// TIA Portal V18 export
ORGANIZATION_BLOCK "Status Monitor"   // OB127, LAD, ProgramCycle
TITLE = Main Control block
{ S7_Optimized_Access := 'TRUE' }
AUTHOR : HenriP
VERSION : 0.1
// stored: AutoNumber true, IsIECCheckEnabled false, SetENOAutomatically false
   VAR_INPUT
      Initial_Call : Bool;   // Initial call of this OB
      Remanence : Bool;   // =True, if remanent data are available
   END_VAR
   VAR_TEMP
      ClearError : Bool;
   END_VAR
   VAR_TEMP   // added for the SCL form of the ladder/FBD networks
      _w1 : Bool;
   END_VAR
BEGIN

REGION Network 1: Monitor
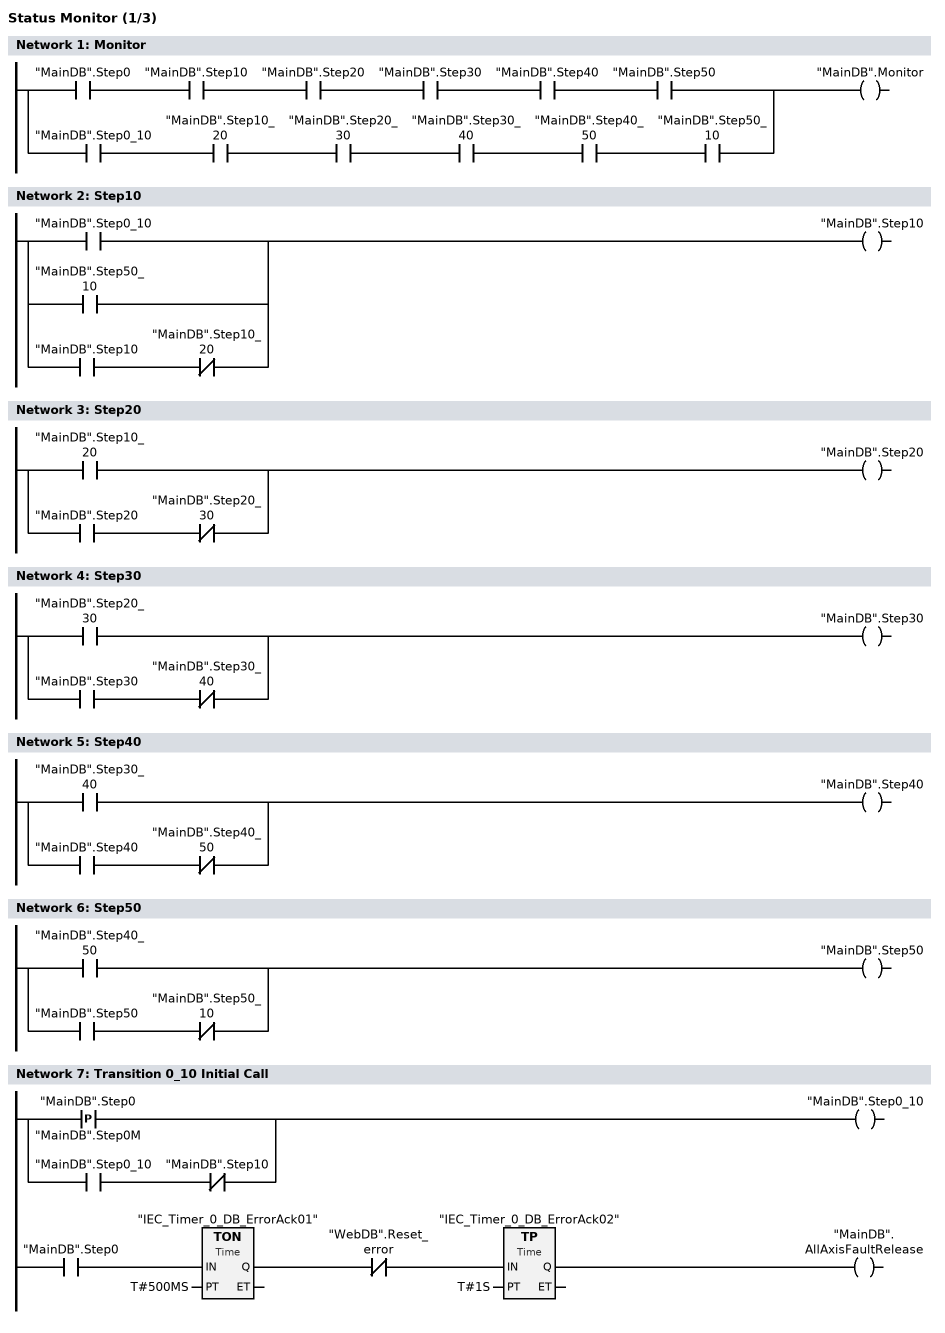
   RUNG wire#powerrail
      Contact( "MainDB".Step0 )
      Contact( "MainDB".Step10 )
      Contact( "MainDB".Step20 )
      Contact( "MainDB".Step30 )
      Contact( "MainDB".Step40 )
      Contact( "MainDB".Step50 )
      wire#w1
      Coil( "MainDB".Monitor )
   END_RUNG
   RUNG wire#powerrail
      Contact( "MainDB".Step0_10 )
      Contact( "MainDB".Step10_20 )
      Contact( "MainDB".Step20_30 )
      Contact( "MainDB".Step30_40 )
      Contact( "MainDB".Step40_50 )
      Contact( "MainDB".Step50_10 )
   END_RUNG wire#w1
   // the same network as SCL:
   "MainDB".Monitor := ("MainDB".Step0 AND "MainDB".Step10 AND "MainDB".Step20 AND "MainDB".Step30 AND "MainDB".Step40 AND "MainDB".Step50) OR ("MainDB".Step0_10 AND "MainDB".Step10_20 AND "MainDB".Step20_30 AND "MainDB".Step30_40 AND "MainDB".Step40_50 AND "MainDB".Step50_10);
END_REGION

REGION Network 2: Step10
   RUNG wire#powerrail
      Contact( "MainDB".Step0_10 )
      wire#w1
      Coil( "MainDB".Step10 )
   END_RUNG
   RUNG wire#powerrail
      Contact( "MainDB".Step50_10 )
   END_RUNG wire#w1
   RUNG wire#powerrail
      Contact( "MainDB".Step10 )
      I_Contact( "MainDB".Step10_20 )
   END_RUNG wire#w1
   // the same network as SCL:
   "MainDB".Step10 := "MainDB".Step0_10 OR "MainDB".Step50_10 OR ("MainDB".Step10 AND NOT "MainDB".Step10_20);
END_REGION

REGION Network 3: Step20
   RUNG wire#powerrail
      Contact( "MainDB".Step10_20 )
      wire#w1
      Coil( "MainDB".Step20 )
   END_RUNG
   RUNG wire#powerrail
      Contact( "MainDB".Step20 )
      I_Contact( "MainDB".Step20_30 )
   END_RUNG wire#w1
   // the same network as SCL:
   "MainDB".Step20 := "MainDB".Step10_20 OR ("MainDB".Step20 AND NOT "MainDB".Step20_30);
END_REGION

REGION Network 4: Step30
   RUNG wire#powerrail
      Contact( "MainDB".Step20_30 )
      wire#w1
      Coil( "MainDB".Step30 )
   END_RUNG
   RUNG wire#powerrail
      Contact( "MainDB".Step30 )
      I_Contact( "MainDB".Step30_40 )
   END_RUNG wire#w1
   // the same network as SCL:
   "MainDB".Step30 := "MainDB".Step20_30 OR ("MainDB".Step30 AND NOT "MainDB".Step30_40);
END_REGION

REGION Network 5: Step40
   RUNG wire#powerrail
      Contact( "MainDB".Step30_40 )
      wire#w1
      Coil( "MainDB".Step40 )
   END_RUNG
   RUNG wire#powerrail
      Contact( "MainDB".Step40 )
      I_Contact( "MainDB".Step40_50 )
   END_RUNG wire#w1
   // the same network as SCL:
   "MainDB".Step40 := "MainDB".Step30_40 OR ("MainDB".Step40 AND NOT "MainDB".Step40_50);
END_REGION

REGION Network 6: Step50
   RUNG wire#powerrail
      Contact( "MainDB".Step40_50 )
      wire#w1
      Coil( "MainDB".Step50 )
   END_RUNG
   RUNG wire#powerrail
      Contact( "MainDB".Step50 )
      I_Contact( "MainDB".Step50_10 )
   END_RUNG wire#w1
   // the same network as SCL:
   "MainDB".Step50 := "MainDB".Step40_50 OR ("MainDB".Step50 AND NOT "MainDB".Step50_10);
END_REGION

REGION Network 7: Transition 0_10 Initial Call
   RUNG wire#powerrail
      P_Contact(operand := "MainDB".Step0, bit := "MainDB".Step0M)
      wire#w1
      Coil( "MainDB".Step0_10 )
   END_RUNG
   RUNG wire#powerrail
      Contact( "MainDB".Step0_10 )
      I_Contact( "MainDB".Step10 )
   END_RUNG wire#w1
   RUNG wire#powerrail
      Contact( "MainDB".Step0 )
      { S7_Templates := "time_type := Time" } "IEC_Timer_0_DB_ErrorAck01".TON(pt := T#500MS, et =>)
      I_Contact( "WebDB".Reset_error )
      { S7_Templates := "time_type := Time" } "IEC_Timer_0_DB_ErrorAck02".TP(pt := T#1S, et =>)
      Coil( "MainDB".AllAxisFaultRelease )
   END_RUNG
   // the same network as SCL:
   #_w1 := "MainDB".Step0 AND NOT "MainDB".Step0M;   // rising edge of "MainDB".Step0
   "MainDB".Step0M := "MainDB".Step0;
   "MainDB".Step0_10 := #_w1 OR ("MainDB".Step0_10 AND NOT "MainDB".Step10);
   "IEC_Timer_0_DB_ErrorAck01".TON(IN := "MainDB".Step0, PT := T#500MS);
   "IEC_Timer_0_DB_ErrorAck02".TP(IN := "IEC_Timer_0_DB_ErrorAck01".Q AND NOT "WebDB".Reset_error, PT := T#1S);
   "MainDB".AllAxisFaultRelease := "IEC_Timer_0_DB_ErrorAck02".Q;
END_REGION

REGION Network 8: Transition10-20 Check PLC Operating State -> Wait Ready
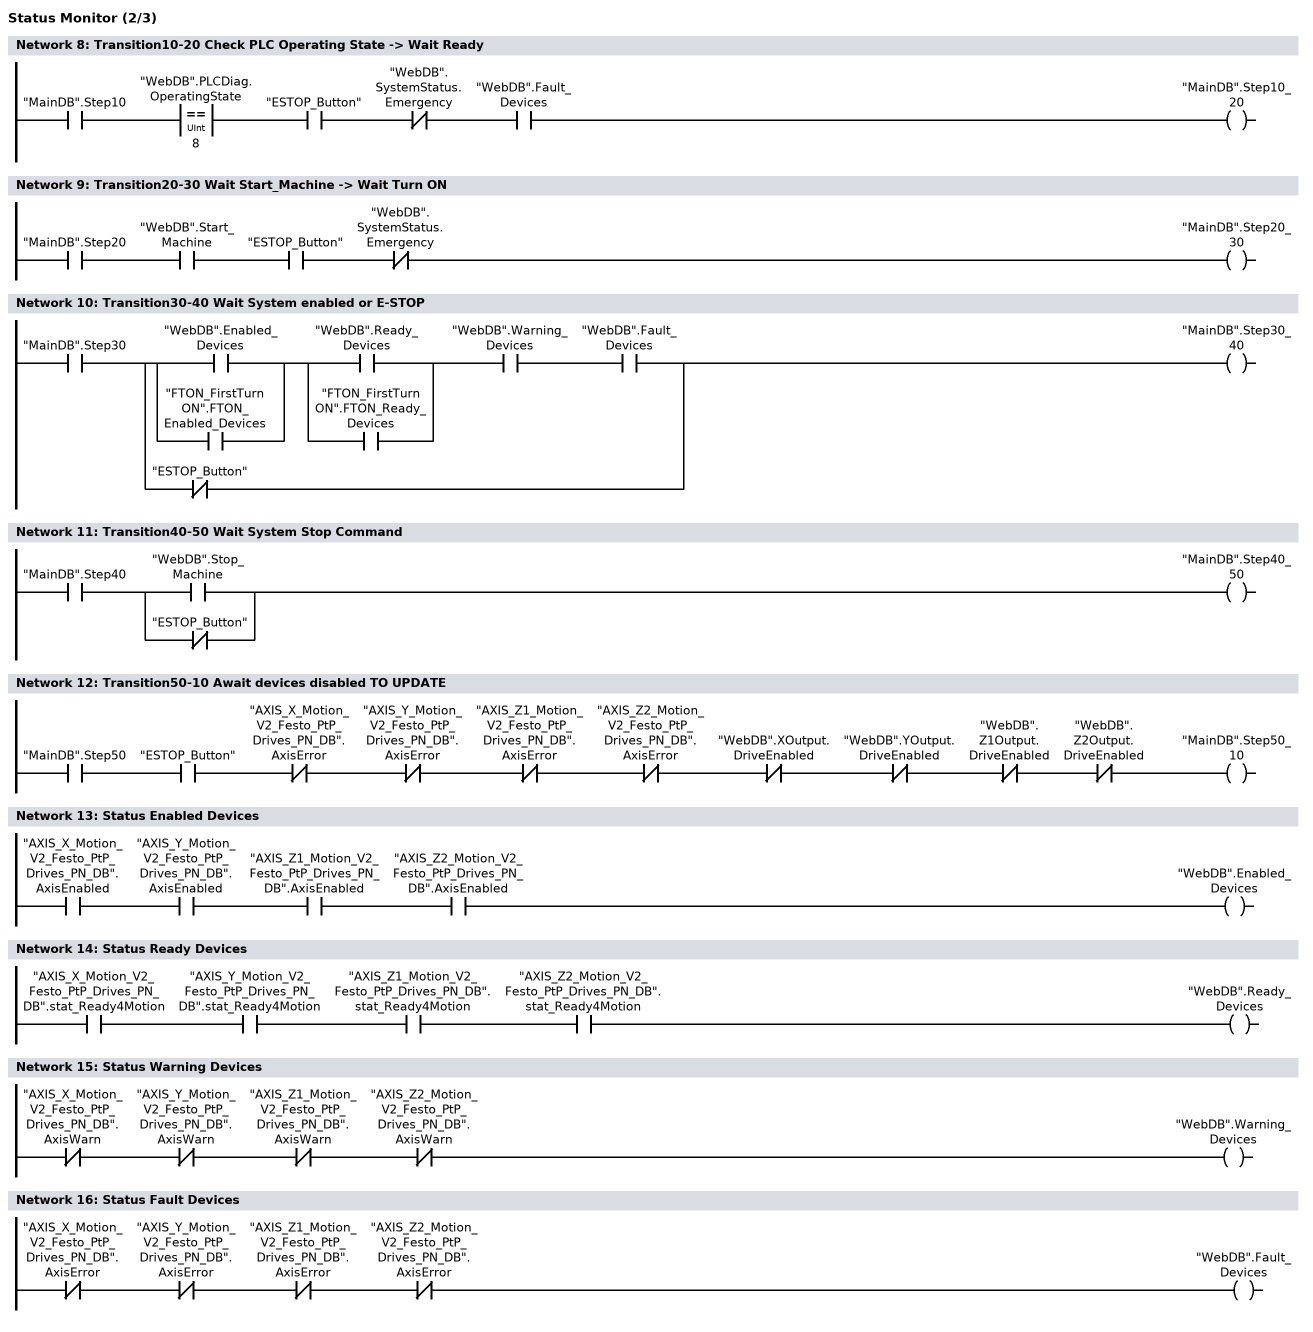
   RUNG wire#powerrail
      Contact( "MainDB".Step10 )
      { S7_Templates := "SrcType := UInt" } EQ_Contact(in1 := "WebDB".PLCDiag.OperatingState, in2 := 8)
      Contact( "ESTOP_Button" )
      I_Contact( "WebDB".SystemStatus.Emergency )
      Contact( "WebDB".Fault_Devices )
      Coil( "MainDB".Step10_20 )
   END_RUNG
   // the same network as SCL:
   "MainDB".Step10_20 := "MainDB".Step10 AND ("WebDB".PLCDiag.OperatingState = 8) AND "ESTOP_Button" AND NOT "WebDB".SystemStatus.Emergency AND "WebDB".Fault_Devices;
END_REGION

REGION Network 9: Transition20-30 Wait Start_Machine -> Wait Turn ON
   RUNG wire#powerrail
      Contact( "MainDB".Step20 )
      Contact( "WebDB".Start_Machine )
      Contact( "ESTOP_Button" )
      I_Contact( "WebDB".SystemStatus.Emergency )
      Coil( "MainDB".Step20_30 )
   END_RUNG
   // the same network as SCL:
   "MainDB".Step20_30 := "MainDB".Step20 AND "WebDB".Start_Machine AND "ESTOP_Button" AND NOT "WebDB".SystemStatus.Emergency;
END_REGION

REGION Network 10: Transition30-40 Wait System enabled or E-STOP
   RUNG wire#powerrail
      Contact( "MainDB".Step30 )
      wire#w1
      Contact( "WebDB".Enabled_Devices )
      wire#w2
      Contact( "WebDB".Ready_Devices )
      wire#w3
      Contact( "WebDB".Warning_Devices )
      Contact( "WebDB".Fault_Devices )
      wire#w4
      Coil( "MainDB".Step30_40 )
   END_RUNG
   RUNG wire#w1
      Contact( "FTON_FirstTurnON".FTON_Enabled_Devices )
   END_RUNG wire#w2
   RUNG wire#w2
      Contact( "FTON_FirstTurnON".FTON_Ready_Devices )
   END_RUNG wire#w3
   RUNG wire#w1
      I_Contact( "ESTOP_Button" )
   END_RUNG wire#w4
   // the same network as SCL:
   "MainDB".Step30_40 := "MainDB".Step30 AND ((("WebDB".Enabled_Devices OR "FTON_FirstTurnON".FTON_Enabled_Devices) AND ("WebDB".Ready_Devices OR "FTON_FirstTurnON".FTON_Ready_Devices) AND "WebDB".Warning_Devices AND "WebDB".Fault_Devices) OR NOT "ESTOP_Button");
END_REGION

REGION Network 11: Transition40-50 Wait System Stop Command
   RUNG wire#powerrail
      Contact( "MainDB".Step40 )
      wire#w1
      Contact( "WebDB".Stop_Machine )
      wire#w2
      Coil( "MainDB".Step40_50 )
   END_RUNG
   RUNG wire#w1
      I_Contact( "ESTOP_Button" )
   END_RUNG wire#w2
   // the same network as SCL:
   "MainDB".Step40_50 := "MainDB".Step40 AND ("WebDB".Stop_Machine OR NOT "ESTOP_Button");
END_REGION

REGION Network 12: Transition50-10 Await devices disabled TO UPDATE
   RUNG wire#powerrail
      Contact( "MainDB".Step50 )
      Contact( "ESTOP_Button" )
      I_Contact( "AXIS_X_Motion_V2_Festo_PtP_Drives_PN_DB".AxisError )
      I_Contact( "AXIS_Y_Motion_V2_Festo_PtP_Drives_PN_DB".AxisError )
      I_Contact( "AXIS_Z1_Motion_V2_Festo_PtP_Drives_PN_DB".AxisError )
      I_Contact( "AXIS_Z2_Motion_V2_Festo_PtP_Drives_PN_DB".AxisError )
      I_Contact( "WebDB".XOutput.DriveEnabled )
      I_Contact( "WebDB".YOutput.DriveEnabled )
      I_Contact( "WebDB".Z1Output.DriveEnabled )
      I_Contact( "WebDB".Z2Output.DriveEnabled )
      Coil( "MainDB".Step50_10 )
   END_RUNG
   // the same network as SCL:
   "MainDB".Step50_10 := "MainDB".Step50 AND "ESTOP_Button" AND NOT "AXIS_X_Motion_V2_Festo_PtP_Drives_PN_DB".AxisError AND NOT "AXIS_Y_Motion_V2_Festo_PtP_Drives_PN_DB".AxisError AND NOT "AXIS_Z1_Motion_V2_Festo_PtP_Drives_PN_DB".AxisError AND NOT "AXIS_Z2_Motion_V2_Festo_PtP_Drives_PN_DB".AxisError AND NOT "WebDB".XOutput.DriveEnabled AND NOT "WebDB".YOutput.DriveEnabled AND NOT "WebDB".Z1Output.DriveEnabled AND NOT "WebDB".Z2Output.DriveEnabled;
END_REGION

REGION Network 13: Status Enabled Devices
   RUNG wire#powerrail
      Contact( "AXIS_X_Motion_V2_Festo_PtP_Drives_PN_DB".AxisEnabled )
      Contact( "AXIS_Y_Motion_V2_Festo_PtP_Drives_PN_DB".AxisEnabled )
      Contact( "AXIS_Z1_Motion_V2_Festo_PtP_Drives_PN_DB".AxisEnabled )
      Contact( "AXIS_Z2_Motion_V2_Festo_PtP_Drives_PN_DB".AxisEnabled )
      Coil( "WebDB".Enabled_Devices )
   END_RUNG
   // the same network as SCL:
   "WebDB".Enabled_Devices := "AXIS_X_Motion_V2_Festo_PtP_Drives_PN_DB".AxisEnabled AND "AXIS_Y_Motion_V2_Festo_PtP_Drives_PN_DB".AxisEnabled AND "AXIS_Z1_Motion_V2_Festo_PtP_Drives_PN_DB".AxisEnabled AND "AXIS_Z2_Motion_V2_Festo_PtP_Drives_PN_DB".AxisEnabled;
END_REGION

REGION Network 14: Status Ready Devices
   RUNG wire#powerrail
      Contact( "AXIS_X_Motion_V2_Festo_PtP_Drives_PN_DB".stat_Ready4Motion )
      Contact( "AXIS_Y_Motion_V2_Festo_PtP_Drives_PN_DB".stat_Ready4Motion )
      Contact( "AXIS_Z1_Motion_V2_Festo_PtP_Drives_PN_DB".stat_Ready4Motion )
      Contact( "AXIS_Z2_Motion_V2_Festo_PtP_Drives_PN_DB".stat_Ready4Motion )
      Coil( "WebDB".Ready_Devices )
   END_RUNG
   // the same network as SCL:
   "WebDB".Ready_Devices := "AXIS_X_Motion_V2_Festo_PtP_Drives_PN_DB".stat_Ready4Motion AND "AXIS_Y_Motion_V2_Festo_PtP_Drives_PN_DB".stat_Ready4Motion AND "AXIS_Z1_Motion_V2_Festo_PtP_Drives_PN_DB".stat_Ready4Motion AND "AXIS_Z2_Motion_V2_Festo_PtP_Drives_PN_DB".stat_Ready4Motion;
END_REGION

REGION Network 15: Status Warning Devices
   RUNG wire#powerrail
      I_Contact( "AXIS_X_Motion_V2_Festo_PtP_Drives_PN_DB".AxisWarn )
      I_Contact( "AXIS_Y_Motion_V2_Festo_PtP_Drives_PN_DB".AxisWarn )
      I_Contact( "AXIS_Z1_Motion_V2_Festo_PtP_Drives_PN_DB".AxisWarn )
      I_Contact( "AXIS_Z2_Motion_V2_Festo_PtP_Drives_PN_DB".AxisWarn )
      Coil( "WebDB".Warning_Devices )
   END_RUNG
   // the same network as SCL:
   "WebDB".Warning_Devices := NOT "AXIS_X_Motion_V2_Festo_PtP_Drives_PN_DB".AxisWarn AND NOT "AXIS_Y_Motion_V2_Festo_PtP_Drives_PN_DB".AxisWarn AND NOT "AXIS_Z1_Motion_V2_Festo_PtP_Drives_PN_DB".AxisWarn AND NOT "AXIS_Z2_Motion_V2_Festo_PtP_Drives_PN_DB".AxisWarn;
END_REGION

REGION Network 16: Status Fault Devices
   RUNG wire#powerrail
      I_Contact( "AXIS_X_Motion_V2_Festo_PtP_Drives_PN_DB".AxisError )
      I_Contact( "AXIS_Y_Motion_V2_Festo_PtP_Drives_PN_DB".AxisError )
      I_Contact( "AXIS_Z1_Motion_V2_Festo_PtP_Drives_PN_DB".AxisError )
      I_Contact( "AXIS_Z2_Motion_V2_Festo_PtP_Drives_PN_DB".AxisError )
      Coil( "WebDB".Fault_Devices )
   END_RUNG
   // the same network as SCL:
   "WebDB".Fault_Devices := NOT "AXIS_X_Motion_V2_Festo_PtP_Drives_PN_DB".AxisError AND NOT "AXIS_Y_Motion_V2_Festo_PtP_Drives_PN_DB".AxisError AND NOT "AXIS_Z1_Motion_V2_Festo_PtP_Drives_PN_DB".AxisError AND NOT "AXIS_Z2_Motion_V2_Festo_PtP_Drives_PN_DB".AxisError;
END_REGION

REGION Network 17: Emergency button is active
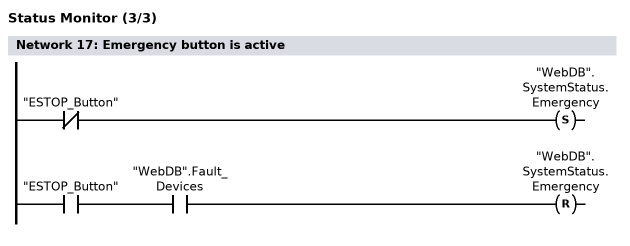
   RUNG wire#powerrail
      I_Contact( "ESTOP_Button" )
      S_Coil( "WebDB".SystemStatus.Emergency )
   END_RUNG
   RUNG wire#powerrail
      Contact( "ESTOP_Button" )
      Contact( "WebDB".Fault_Devices )
      R_Coil( "WebDB".SystemStatus.Emergency )
   END_RUNG
   // the same network as SCL:
   IF NOT "ESTOP_Button" THEN "WebDB".SystemStatus.Emergency := TRUE; END_IF;
   IF "ESTOP_Button" AND "WebDB".Fault_Devices THEN "WebDB".SystemStatus.Emergency := FALSE; END_IF;
END_REGION
END_ORGANIZATION_BLOCK
